{region '#Template'}
	{attribute 'Category' := 'AC'}
	{attribute 'Version' := '0.0.1.0'}
	{attribute 'Tags' := 'AC, Plant, AHU, Air handling unit'}
	{attribute 'Description' := 'Lüftungsanlage	// Air handling unit'}
{endregion}
FUNCTION_BLOCK FB_BA_AHU_1St_PrHtr_ErcPl_Col EXTENDS FB_BA_View
VAR_INPUT CONSTANT	
	TOuA					: FB_BA_SensorAnalog_IO;			
	TExhA					: FB_BA_SensorAnalog_IO;	
	TSuA					: FB_BA_SensorAnalog_IO;	
	TExtA					: FB_BA_SensorAnalog_IO;								
	TRm						: FB_BA_SensorAnalog_IO;	
	DiffPrssOuAFilt			: FB_BA_SensorAnalog_IO;											
	FiltOuAMonit			: FB_BA_Hys_21;							
	DiffPrssExtAFilt		: FB_BA_SensorAnalog_IO;				
	FiltExtAMonit			: FB_BA_Hys_21;	
	SumNgtCol				: FB_BA_AC_SumNgtCol;	
	OpMod					: FB_BA_AC_OpMod1St;	
	OuADmp					: FB_BA_Dmp2P;	
	SuAPrss					: FB_BA_SensorAnalog_IO;	
	SuADiffPrss				: FB_BA_SensorAnalog_IO;		
	SuAFan					: FB_BA_MotCtlExt;	
	SuADiffPrssMonit		: FB_BA_FdbAnalog;								
	ExhADmp					: FB_BA_Dmp2P;	
	ExtAPrss				: FB_BA_SensorAnalog_IO;	
	ExtADiffPrss			: FB_BA_SensorAnalog_IO;		
	ExtAFan					: FB_BA_MotCtlExt;								
	ExtADiffPrssMonit		: FB_BA_FdbAnalog;
	SpTRm					: FB_BA_AC_SpTRm_01;	
	TCasCtrl				: FB_BA_AC_TCasCtrl_01;										 								
	TSeqLink				: FB_BA_SequenceLink;
	PreHtr					: FB_BA_AC_PreHtr;	
	Erc						: FB_BA_AC_ErcPl_02;								
	Col						: FB_BA_AC_ColT_02;								
	PlantCtrl				: FB_BA_PlantCtrl;							
	GeneralSettings			: FB_BA_RawSubscriber;
	stGeneralSettings		: ST_BA_GeneralSettings;
END_VAR	
VAR
	PlantLock				: FB_BA_PlantLock	:= (iParent := THIS^);	
	
	PlantControlStatus   	:FB_BA_Label2x :=(iAggregate:=LblControl.PlantControl,		iFunction:=LblFunctions.Status);
	TSequenceControlStatus  :FB_BA_Label2x :=(iAggregate:=LblControl.TSequenceControl,	iFunction:=LblFunctions.Status);	
END_VAR
VAR // added by the converter: edge detectors and wires of the graphical bodies
    _w1 : ANY;
END_VAR

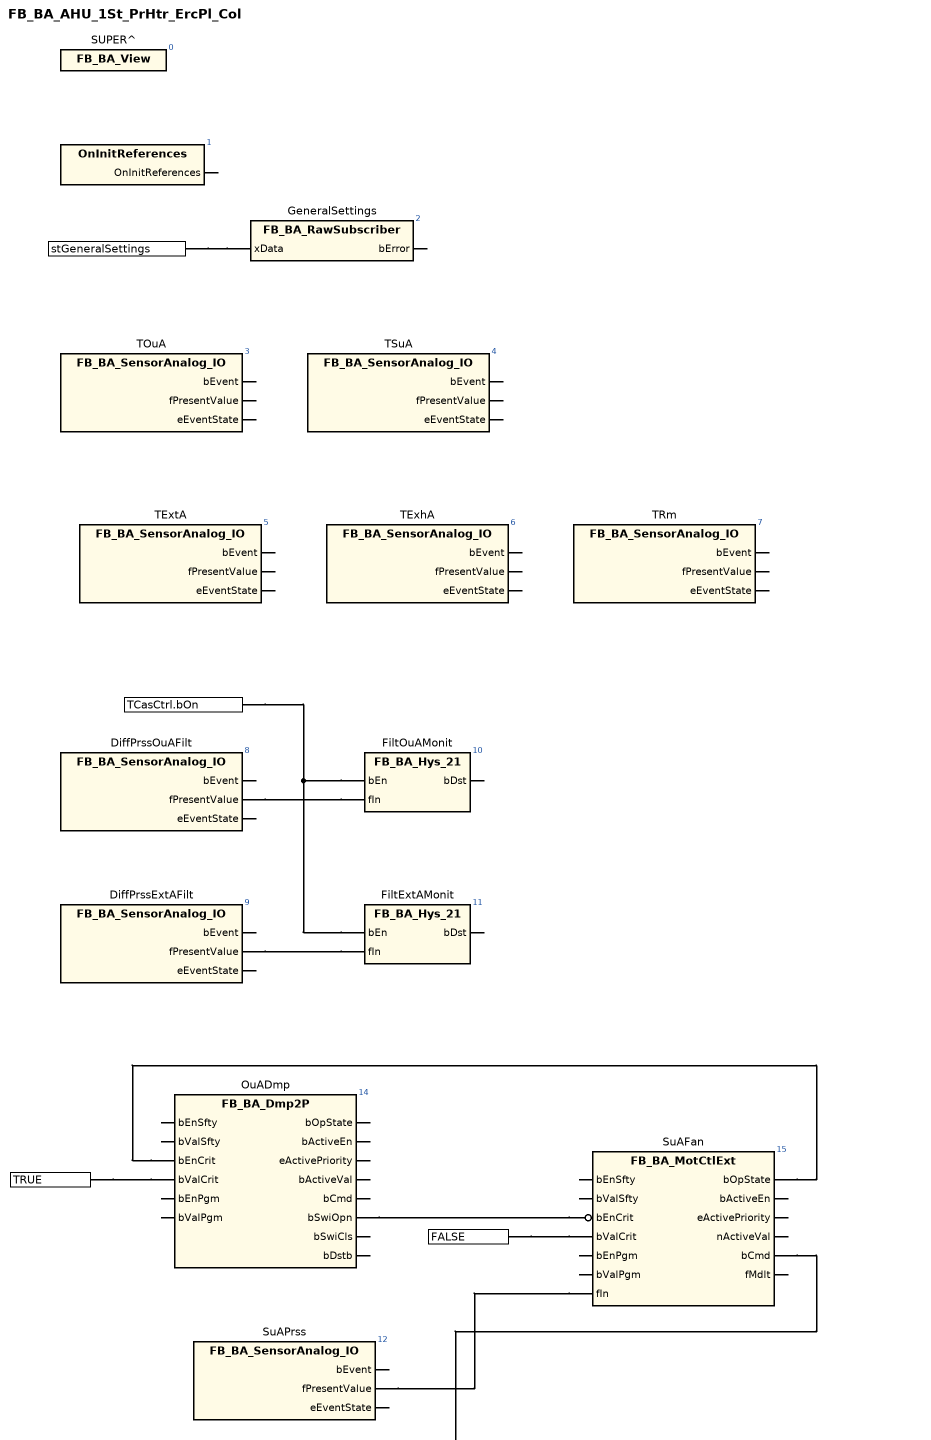
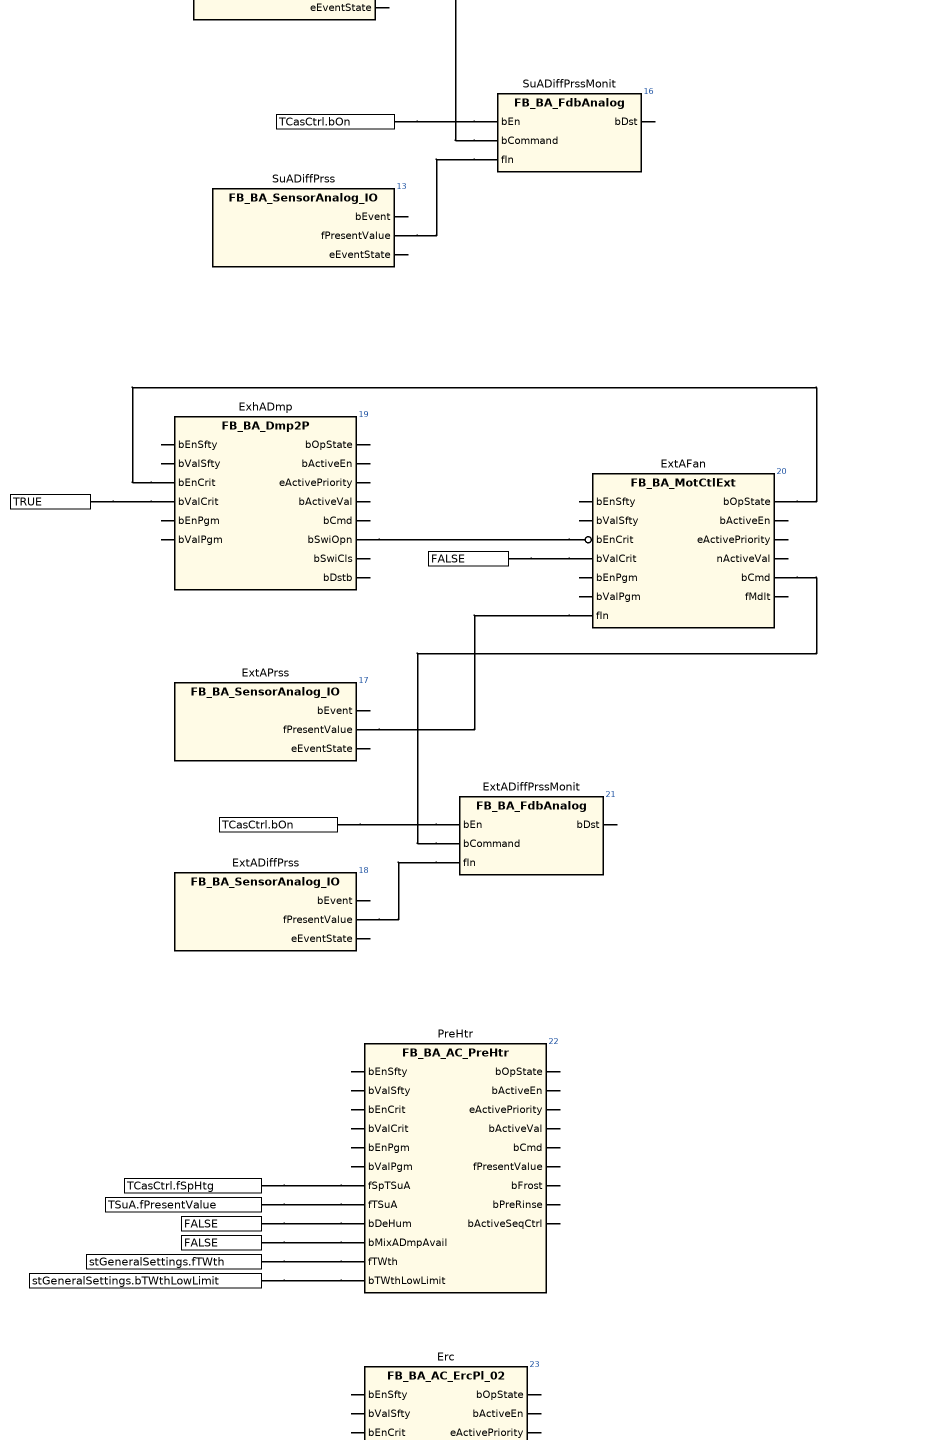
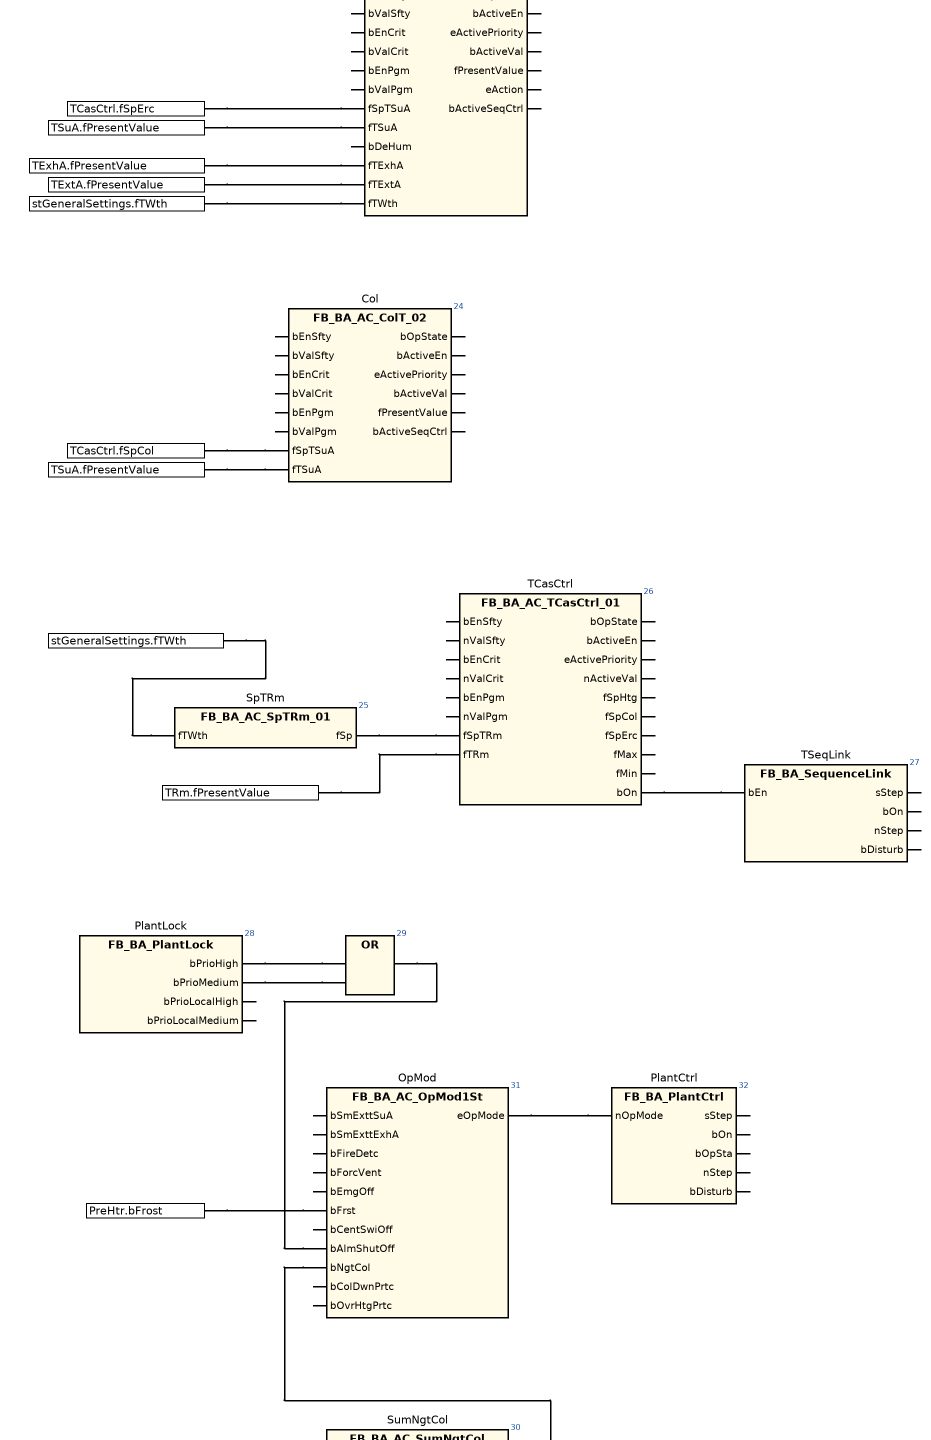
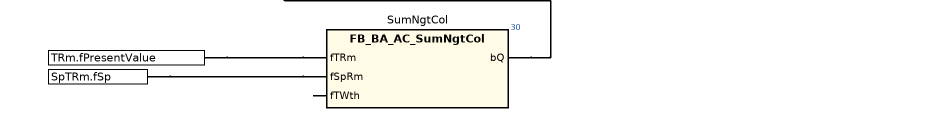
SUPER^(); // FB_BA_View
OnInitReferences();
GeneralSettings(xData := stGeneralSettings); // FB_BA_RawSubscriber
TOuA(); // FB_BA_SensorAnalog_IO
TSuA(); // FB_BA_SensorAnalog_IO
TExtA(); // FB_BA_SensorAnalog_IO
TExhA(); // FB_BA_SensorAnalog_IO
TRm(); // FB_BA_SensorAnalog_IO
DiffPrssOuAFilt(); // FB_BA_SensorAnalog_IO
DiffPrssExtAFilt(); // FB_BA_SensorAnalog_IO
FiltOuAMonit(bEn := TCasCtrl.bOn, fIn := DiffPrssOuAFilt.fPresentValue); // FB_BA_Hys_21
FiltExtAMonit(bEn := TCasCtrl.bOn, fIn := DiffPrssExtAFilt.fPresentValue); // FB_BA_Hys_21
SuAPrss(); // FB_BA_SensorAnalog_IO
SuADiffPrss(); // FB_BA_SensorAnalog_IO
OuADmp(bEnCrit := SuAFan.bOpState, bValCrit := TRUE); // FB_BA_Dmp2P
SuAFan(bEnCrit := NOT OuADmp.bSwiOpn, bValCrit := FALSE, fIn := SuAPrss.fPresentValue); // FB_BA_MotCtlExt
SuADiffPrssMonit(bEn := TCasCtrl.bOn, bCommand := SuAFan.bCmd, fIn := SuADiffPrss.fPresentValue); // FB_BA_FdbAnalog
ExtAPrss(); // FB_BA_SensorAnalog_IO
ExtADiffPrss(); // FB_BA_SensorAnalog_IO
ExhADmp(bEnCrit := ExtAFan.bOpState, bValCrit := TRUE); // FB_BA_Dmp2P
ExtAFan(bEnCrit := NOT ExhADmp.bSwiOpn, bValCrit := FALSE, fIn := ExtAPrss.fPresentValue); // FB_BA_MotCtlExt
ExtADiffPrssMonit(bEn := TCasCtrl.bOn, bCommand := ExtAFan.bCmd, fIn := ExtADiffPrss.fPresentValue); // FB_BA_FdbAnalog
PreHtr(
    fSpTSuA := TCasCtrl.fSpHtg,
    fTSuA := TSuA.fPresentValue,
    bDeHum := FALSE,
    bMixADmpAvail := FALSE,
    fTWth := stGeneralSettings.fTWth,
    bTWthLowLimit := stGeneralSettings.bTWthLowLimit); // FB_BA_AC_PreHtr
Erc(
    fSpTSuA := TCasCtrl.fSpErc,
    fTSuA := TSuA.fPresentValue,
    fTExhA := TExhA.fPresentValue,
    fTExtA := TExtA.fPresentValue,
    fTWth := stGeneralSettings.fTWth); // FB_BA_AC_ErcPl_02
Col(fSpTSuA := TCasCtrl.fSpCol, fTSuA := TSuA.fPresentValue); // FB_BA_AC_ColT_02
SpTRm(fTWth := stGeneralSettings.fTWth); // FB_BA_AC_SpTRm_01
TCasCtrl(fSpTRm := SpTRm.fSp, fTRm := TRm.fPresentValue); // FB_BA_AC_TCasCtrl_01
TSeqLink(bEn := TCasCtrl.bOn); // FB_BA_SequenceLink
PlantLock(); // FB_BA_PlantLock
_w1 := PlantLock.bPrioHigh OR PlantLock.bPrioMedium;
SumNgtCol(fTRm := TRm.fPresentValue, fSpRm := SpTRm.fSp); // FB_BA_AC_SumNgtCol
OpMod(bFrst := PreHtr.bFrost, bAlmShutOff := _w1, bNgtCol := SumNgtCol.bQ); // FB_BA_AC_OpMod1St
PlantCtrl(nOpMode := OpMod.eOpMode); // FB_BA_PlantCtrl

METHOD FB_init : BOOL
VAR_INPUT
	bInitRetains : BOOL; // if TRUE, the retain variables are initialized (warm start / cold start)
	bInCopyCode : BOOL;  // if TRUE, the instance afterwards gets moved into the copy code (online change)
END_VAR
TOuA.iParent								:= THIS^;		
TOuA.iLabel 								:= LblCmpAC.AHU_TOuA;	
TOuA.sObjectName							:= '{Idx=01}';	
TOuA.eDPADMode								:= E_BA_DPADMode.eInclude;										
TOuA.MV.eUnit								:= E_BA_Unit.eTemperature_DegreesCelsius;
TOuA.MV.eEnPlantLock						:= E_BA_LockPriority.eNoLock;
TOuA.MV.fResolution 						:= 0.01;
TOuA.MV.fScaleOffset 						:= 0; 

TExhA.iParent								:= THIS^;		
TExhA.iLabel 								:= LblCmpAC.AHU_TExhA;	
TExhA.sObjectName							:= '{Idx=01}';												
TExhA.eDPADMode								:= E_BA_DPADMode.eInclude;										
TExhA.MV.eUnit								:= E_BA_Unit.eTemperature_DegreesCelsius;
TExhA.MV.eEnPlantLock						:= E_BA_LockPriority.eNoLock;
TExhA.MV.fResolution 						:= 0.01;
TExhA.MV.fScaleOffset 						:= 0; 

TSuA.iParent								:= THIS^;		
TSuA.iLabel 								:= LblCmpAC.AHU_TSuA;	
TSuA.sObjectName							:= '{Idx=01}';
TSuA.eDPADMode								:= E_BA_DPADMode.eInclude;										
TSuA.MV.eUnit								:= E_BA_Unit.eTemperature_DegreesCelsius;
TSuA.MV.eEnPlantLock						:= E_BA_LockPriority.eMedium;
TSuA.MV.fResolution 						:= 0.01;
TSuA.MV.fScaleOffset 						:= 0; 

TExtA.iParent								:= THIS^;
TExtA.iLabel 								:= LblCmpAC.AHU_TExtA;	
TExtA.sObjectName							:= '{Idx=01}'; 
TExtA.eDPADMode								:= E_BA_DPADMode.eInclude;										
TExtA.MV.eUnit								:= E_BA_Unit.eTemperature_DegreesCelsius;
TExtA.MV.eEnPlantLock						:= E_BA_LockPriority.eNoLock;
TExtA.MV.fResolution 						:= 0.01;
TExtA.MV.fScaleOffset 						:= 0; 

TRm.iParent									:= THIS^;		
TRm.iLabel 									:= LblCmpAC.AHU_TRm;	
TRm.sObjectName								:= '{Idx=01}';
TRm.eDPADMode								:= E_BA_DPADMode.eInclude;										
TRm.MV.eUnit								:= E_BA_Unit.eTemperature_DegreesCelsius;
TRm.MV.eEnPlantLock							:= E_BA_LockPriority.eNoLock;
TRm.MV.fResolution 							:= 0.01;
TRm.MV.fScaleOffset 						:= 0;

DiffPrssOuAFilt.iParent						:= THIS^;		
DiffPrssOuAFilt.iLabel 						:= LblCmpAC.AHU_DiffPrssOuAFilt;	
DiffPrssOuAFilt.sObjectName					:= '{Idx=03}';												
DiffPrssOuAFilt.eDPADMode					:= E_BA_DPADMode.eInclude;										
DiffPrssOuAFilt.MV.eUnit					:= E_BA_Unit.ePressure_Pascals;
DiffPrssOuAFilt.MV.eEnPlantLock				:= E_BA_LockPriority.eNoLock;
DiffPrssOuAFilt.MV.fResolution 				:= 0.03051851;
DiffPrssOuAFilt.MV.fScaleOffset 			:= 0; 

FiltOuAMonit.iParent						:= THIS^;
FiltOuAMonit.iLabel							:= LblCmpAC.AHU_FiltOuAMonit;
FiltOuAMonit.sObjectName					:= '{Idx=01}';										 
FiltOuAMonit.eDPADMode						:= E_BA_DPADMode.eInclude;
FiltOuAMonit.DstMainAlarm.eEnPlantLock		:= E_BA_LockPriority.eMedium;

DiffPrssExtAFilt.iParent					:= THIS^;		
DiffPrssExtAFilt.iLabel 					:= LblCmpAC.AHU_DiffPrssExtAFilt;	
DiffPrssExtAFilt.sObjectName				:= '{Idx=04}';
DiffPrssExtAFilt.eDPADMode					:= E_BA_DPADMode.eInclude;										
DiffPrssExtAFilt.MV.eUnit					:= E_BA_Unit.ePressure_Pascals;
DiffPrssExtAFilt.MV.eEnPlantLock			:= E_BA_LockPriority.eNoLock;
DiffPrssExtAFilt.MV.fResolution 			:= 0.03051851;
DiffPrssExtAFilt.MV.fScaleOffset 			:= 0; 

FiltExtAMonit.iParent						:= THIS^;
FiltExtAMonit.iLabel						:= LblCmpAC.AHU_FiltExtAMonit;
FiltExtAMonit.sObjectName					:= '{Idx=02}';										 
FiltExtAMonit.eDPADMode						:= E_BA_DPADMode.eInclude;
FiltExtAMonit.DstMainAlarm.eEnPlantLock		:= E_BA_LockPriority.eMedium;

SumNgtCol.iParent							:= THIS^;
SumNgtCol.iLabel							:= LblCmpAC.AHU_SumNgtCol;
SumNgtCol.sObjectName						:= '{Idx=01}';										 
SumNgtCol.eDPADMode							:= E_BA_DPADMode.eInclude;								

OpMod.iParent								:= THIS^;
OpMod.iLabel								:= LblCmpAC.AHU_OpMod;
OpMod.sObjectName							:= '{Idx=01}';										 
OpMod.eDPADMode								:= E_BA_DPADMode.eInclude;								

OuADmp.iParent								:= THIS^;
OuADmp.iLabel								:= LblCmpAC.AHU_OuADmp;
OuADmp.sObjectName							:= '{Idx=01}';										 
OuADmp.eDPADMode							:= E_BA_DPADMode.eInclude;								

SuAPrss.iParent								:= THIS^;		
SuAPrss.iLabel 								:= LblCmpAC.AHU_SuAPrss;	
SuAPrss.sObjectName							:= '{Idx=01}';
SuAPrss.eDPADMode							:= E_BA_DPADMode.eInclude;																						
SuAPrss.MV.eUnit							:= E_BA_Unit.ePressure_Pascals;
SuAPrss.MV.eEnPlantLock						:= E_BA_LockPriority.eNoLock;
SuAPrss.MV.fResolution 						:= 0.03051851;
SuAPrss.MV.fScaleOffset 					:= 0;

SuADiffPrss.iParent							:= THIS^;		
SuADiffPrss.iLabel 							:= LblCmpAC.AHU_SuADiffPrss;	
SuADiffPrss.sObjectName						:= '{Idx=01}';
SuADiffPrss.eDPADMode						:= E_BA_DPADMode.eInclude;																						
SuADiffPrss.MV.eUnit						:= E_BA_Unit.ePressure_Pascals;
SuADiffPrss.MV.eEnPlantLock					:= E_BA_LockPriority.eNoLock;
SuADiffPrss.MV.fResolution 					:= 0.03051851;
SuADiffPrss.MV.fScaleOffset 				:= 0; 

SuAFan.iParent								:= THIS^;
SuAFan.iLabel								:= LblCmpAC.AHU_SuAFan;
SuAFan.sObjectName							:= '{Idx=01}';										 
SuAFan.eDPADMode							:= E_BA_DPADMode.eInclude;								

SuADiffPrssMonit.iParent					:= THIS^;
SuADiffPrssMonit.iLabel						:= LblCmpAC.AHU_SuADiffPrssMonit;
SuADiffPrssMonit.sObjectName				:= '{Idx=01}';										 
SuADiffPrssMonit.eDPADMode					:= E_BA_DPADMode.eInclude;								

ExhADmp.iParent								:= THIS^;
ExhADmp.iLabel								:= LblCmpAC.AHU_ExhADmp;
ExhADmp.sObjectName							:= '{Idx=02}';										 
ExhADmp.eDPADMode							:= E_BA_DPADMode.eInclude;								

ExtAPrss.iParent							:= THIS^;		
ExtAPrss.iLabel 							:= LblCmpAC.AHU_ExtAPrss;	
ExtAPrss.sObjectName						:= '{Idx=01}';												
ExtAPrss.eDPADMode							:= E_BA_DPADMode.eInclude;																						
ExtAPrss.MV.eUnit							:= E_BA_Unit.ePressure_Pascals;
ExtAPrss.MV.eEnPlantLock					:= E_BA_LockPriority.eNoLock;
ExtAPrss.MV.fResolution 					:= 0.03051851;
ExtAPrss.MV.fScaleOffset 					:= 0; 

ExtADiffPrss.iParent						:= THIS^;		
ExtADiffPrss.iLabel 						:= LblCmpAC.AHU_ExtADiffPrss;	
ExtADiffPrss.sObjectName					:= '{Idx=02}';
ExtADiffPrss.eDPADMode						:= E_BA_DPADMode.eInclude;																						
ExtADiffPrss.MV.eUnit						:= E_BA_Unit.ePressure_Pascals;
ExtADiffPrss.MV.eEnPlantLock				:= E_BA_LockPriority.eNoLock;
ExtADiffPrss.MV.fResolution 				:= 0.03051851;
ExtADiffPrss.MV.fScaleOffset 				:= 0; 

ExtAFan.iParent								:= THIS^;
ExtAFan.iLabel								:= LblCmpAC.AHU_ExtAFan;
ExtAFan.sObjectName							:= '{Idx=01}';										 
ExtAFan.eDPADMode							:= E_BA_DPADMode.eInclude;								

ExtADiffPrssMonit.iParent					:= THIS^;
ExtADiffPrssMonit.iLabel					:= LblCmpAC.AHU_ExtADiffPrssMonit;
ExtADiffPrssMonit.sObjectName				:= '{Idx=02}';										 
ExtADiffPrssMonit.eDPADMode					:= E_BA_DPADMode.eInclude;								

SpTRm.iParent								:= THIS^;
SpTRm.iLabel								:= LblCmpAC.AHU_SpTRm;
SpTRm.sObjectName							:= '{Idx=01}';										 
SpTRm.eDPADMode								:= E_BA_DPADMode.eInclude;								

TCasCtrl.iParent							:= THIS^;
TCasCtrl.iLabel								:= LblCmpAC.AHU_TCasCtrl;
TCasCtrl.sObjectName						:= '{Idx=01}';										 
TCasCtrl.eDPADMode							:= E_BA_DPADMode.eInclude;																		 								

TSeqLink.iParent							:= THIS^;
TSeqLink.iLabel								:= LblCmpAC.AHU_TSeqLink;
TSeqLink.sObjectName						:= '{Idx=01,Idx=01}';									
TSeqLink.iReference[1]						:= PreHtr.TSuACtrl.Ctrl;
TSeqLink.iReference[2]						:= Erc.TSuACtrl.Ctrl;
TSeqLink.iReference[3]						:= Col.TSuACtrl.Ctrl;

PreHtr.iParent								:= THIS^;
PreHtr.iLabel								:= LblCmpAC.AHU_PreHtr;
PreHtr.sObjectName							:= '{Idx=01}';										 
PreHtr.eDPADMode							:= E_BA_DPADMode.eIncludeDescription;								

Erc.iParent									:= THIS^;
Erc.iLabel									:= LblCmpAC.AHU_Erc;
Erc.sObjectName								:= '{Idx=01}';										 
Erc.eDPADMode								:= E_BA_DPADMode.eIncludeDescription;																

Col.iParent									:= THIS^;
Col.iLabel									:= LblCmpAC.AHU_Col;
Col.sObjectName								:= '{Idx=01}';										 
Col.eDPADMode								:= E_BA_DPADMode.eIncludeDescription;								

PlantCtrl.iParent							:= THIS^;
PlantCtrl.iLabel							:= LblCmpAC.AHU_PlantCtrl;
PlantCtrl.sObjectName						:= '{Idx=01,Idx=01}';
PlantCtrl.aStateText						:= OpMod.OpModPr.aStateText;	

GeneralSettings.Subject						:= Site.GeneralSettings_Subject;
GeneralSettings.sTarget						:= Site.GeneralSettings_NetId;
END_METHOD

METHOD Init_OffOn : BOOL
// Apply configured states:
(*

WIRD DIESE DEKLARATION HIER BENÖTIGT????
23.02.2021 FP

OpMod.OpModMan.aStateText[1] := Texts.txtAuto;
OpMod.OpModMan.aStateText[2] := Texts.txtOff;
OpMod.OpModMan.aStateText[3] := Texts.txtOn;

OpMod.Sched.aStateText[1] := Texts.txtOff;
OpMod.Sched.aStateText[2] := Texts.txtOn;

OpMod.OpModPr.aStateText[1]		:= Texts.txtOff;
OpMod.OpModPr.aStateText[2]		:= Texts.txtOn;
OpMod.OpModPr.aStateText[3]		:= Texts.txtEmergencyStop;
OpMod.OpModPr.aStateText[4]		:= Texts.txtFrost;
OpMod.OpModPr.aStateText[5]		:= Texts.txtSmokeExtraction_P;
OpMod.OpModPr.aStateText[6]		:= Texts.txtSmokeExtractionSupplyAir;
OpMod.OpModPr.aStateText[7]		:= Texts.txtSmokeExtractionExtractAir;
OpMod.OpModPr.aStateText[8]		:= Texts.txtFire;
OpMod.OpModPr.aStateText[9]		:= Texts.txtNightCooling;
OpMod.OpModPr.aStateText[10]	:= Texts.txtCoolDownProtection;
OpMod.OpModPr.aStateText[11]	:= Texts.txtOverHeatingProtection;
OpMod.OpModPr.aStateText[12]	:= Texts.txtDisturb;
OpMod.OpModPr.aStateText[13]	:= Texts.txtForcedVentilation;
OpMod.OpModPr.aStateText[14]	:= Texts.txtCentralSwitchOff;
*)

// plant operations modes with priorities:
PlantCtrl.AddOperationMode(nOpMode := E_BA_AC_OpMod01.eOff,							ePriority := E_BA_Priority.eProgram);
PlantCtrl.AddOperationMode(nOpMode := E_BA_AC_OpMod01.eOn,							ePriority := E_BA_Priority.eProgram);
PlantCtrl.AddOperationMode(nOpMode := E_BA_AC_OpMod01.eNightCooling,				ePriority := E_BA_Priority.eProgram);
PlantCtrl.AddOperationMode(nOpMode := E_BA_AC_OpMod01.eCoolDownProtection,			ePriority := E_BA_Priority.eProgram);
PlantCtrl.AddOperationMode(nOpMode := E_BA_AC_OpMod01.eOverHeatingProtection,		ePriority := E_BA_Priority.eProgram);
PlantCtrl.AddOperationMode(nOpMode := E_BA_AC_OpMod01.eFrost,						ePriority := E_BA_Priority.eCritical);
PlantCtrl.AddOperationMode(nOpMode := E_BA_AC_OpMod01.eEmergency,					ePriority := E_BA_Priority.eCritical);
PlantCtrl.AddOperationMode(nOpMode := E_BA_AC_OpMod01.eAlarm,						ePriority := E_BA_Priority.eCritical);
PlantCtrl.AddOperationMode(nOpMode := E_BA_AC_OpMod01.eForcedVentilation,			ePriority := E_BA_Priority.eCritical);
PlantCtrl.AddOperationMode(nOpMode := E_BA_AC_OpMod01.eCentralSwitchOff,			ePriority := E_BA_Priority.eCritical);
PlantCtrl.AddOperationMode(nOpMode := E_BA_AC_OpMod01.eSmokeExtractionProgramm,		ePriority := E_BA_Priority.eLifeSafety);
PlantCtrl.AddOperationMode(nOpMode := E_BA_AC_OpMod01.eSmokeExtractionSupplyAir,	ePriority := E_BA_Priority.eLifeSafety);
PlantCtrl.AddOperationMode(nOpMode := E_BA_AC_OpMod01.eSmokeExtractionExhaustAir,	ePriority := E_BA_Priority.eLifeSafety);
PlantCtrl.AddOperationMode(nOpMode := E_BA_AC_OpMod01.eFire, 						ePriority := E_BA_Priority.eLifeSafety);

// Start sequence Step order and parameter
PlantCtrl.AddAggregate(iReference := PreHtr,	bWaitForProcesses := TRUE,	bWaitForEvents := FALSE, tDelayStepDown := T#0S, tDelayStepUp := T#5S);
PlantCtrl.AddAggregate(iReference := OuADmp,	bWaitForProcesses := FALSE, bWaitForEvents := FALSE, tDelayStepDown := T#2S, tDelayStepUp := T#2S);
PlantCtrl.AddAggregate(iReference := ExhADmp,	bWaitForProcesses := FALSE, bWaitForEvents := FALSE, tDelayStepDown := T#2S, tDelayStepUp := T#2S);
PlantCtrl.AddAggregate(iReference := SuAFan,	bWaitForProcesses := FALSE, bWaitForEvents := FALSE, tDelayStepDown := T#2S, tDelayStepUp := T#2S);
PlantCtrl.AddAggregate(iReference := ExtAFan,	bWaitForProcesses := FALSE, bWaitForEvents := FALSE, tDelayStepDown := T#2S, tDelayStepUp := T#2S);
PlantCtrl.AddAggregate(iReference := Erc,		bWaitForProcesses := FALSE, bWaitForEvents := FALSE, tDelayStepDown := T#0S, tDelayStepUp := T#0S);
PlantCtrl.AddAggregate(iReference := Col,		bWaitForProcesses := FALSE, bWaitForEvents := FALSE, tDelayStepDown := T#0S, tDelayStepUp := T#0S);
PlantCtrl.AddAggregate(iReference := TCasCtrl,	bWaitForProcesses := FALSE, bWaitForEvents := FALSE, tDelayStepDown := T#0S, tDelayStepUp := T#0S);

// Apply aggregate operation modes dependant on corresponding plant operation modes:
// [Controlling aggregates]
// release pre-heater depending on plant operation mode 
PlantCtrl.AssignAggregate1x(nPltOpMode := E_BA_AC_OpMod01.eOff,							iAgg1Ref := PreHtr, nAgg1OpMode := TO_UDINT(FALSE));
PlantCtrl.AssignAggregate1x(nPltOpMode := E_BA_AC_OpMod01.eOn,							iAgg1Ref := PreHtr, nAgg1OpMode := TO_UDINT(TRUE));
PlantCtrl.AssignAggregate1x(nPltOpMode := E_BA_AC_OpMod01.eNightCooling,				iAgg1Ref := PreHtr, nAgg1OpMode := TO_UDINT(FALSE));
PlantCtrl.AssignAggregate1x(nPltOpMode := E_BA_AC_OpMod01.eCoolDownProtection,			iAgg1Ref := PreHtr, nAgg1OpMode := TO_UDINT(TRUE));
PlantCtrl.AssignAggregate1x(nPltOpMode := E_BA_AC_OpMod01.eOverHeatingProtection,		iAgg1Ref := PreHtr, nAgg1OpMode := TO_UDINT(FALSE));
PlantCtrl.AssignAggregate1x(nPltOpMode := E_BA_AC_OpMod01.eFrost,						iAgg1Ref := PreHtr, nAgg1OpMode := TO_UDINT(TRUE));
PlantCtrl.AssignAggregate1x(nPltOpMode := E_BA_AC_OpMod01.eEmergency,					iAgg1Ref := PreHtr, nAgg1OpMode := TO_UDINT(FALSE));
PlantCtrl.AssignAggregate1x(nPltOpMode := E_BA_AC_OpMod01.eAlarm,						iAgg1Ref := PreHtr, nAgg1OpMode := TO_UDINT(FALSE));
PlantCtrl.AssignAggregate1x(nPltOpMode := E_BA_AC_OpMod01.eForcedVentilation,			iAgg1Ref := PreHtr, nAgg1OpMode := TO_UDINT(TRUE));
PlantCtrl.AssignAggregate1x(nPltOpMode := E_BA_AC_OpMod01.eCentralSwitchOff,			iAgg1Ref := PreHtr, nAgg1OpMode := TO_UDINT(FALSE));
PlantCtrl.AssignAggregate1x(nPltOpMode := E_BA_AC_OpMod01.eSmokeExtractionProgramm,		iAgg1Ref := PreHtr, nAgg1OpMode := TO_UDINT(TRUE));
PlantCtrl.AssignAggregate1x(nPltOpMode := E_BA_AC_OpMod01.eSmokeExtractionSupplyAir,	iAgg1Ref := PreHtr, nAgg1OpMode := TO_UDINT(TRUE));
PlantCtrl.AssignAggregate1x(nPltOpMode := E_BA_AC_OpMod01.eSmokeExtractionExhaustAir,	iAgg1Ref := PreHtr, nAgg1OpMode := TO_UDINT(FALSE));
PlantCtrl.AssignAggregate1x(nPltOpMode := E_BA_AC_OpMod01.eFire,						iAgg1Ref := PreHtr, nAgg1OpMode := TO_UDINT(FALSE));

// Apply aggregate operation modes dependant on corresponding plant operation modes:
// [Controlling aggregates]
// release Erc depending on plant operation mode 
PlantCtrl.AssignAggregate1x(nPltOpMode := E_BA_AC_OpMod01.eOff,							iAgg1Ref := Erc, nAgg1OpMode := TO_UDINT(FALSE));
PlantCtrl.AssignAggregate1x(nPltOpMode := E_BA_AC_OpMod01.eOn,							iAgg1Ref := Erc, nAgg1OpMode := TO_UDINT(TRUE));
PlantCtrl.AssignAggregate1x(nPltOpMode := E_BA_AC_OpMod01.eNightCooling,				iAgg1Ref := Erc, nAgg1OpMode := TO_UDINT(FALSE));
PlantCtrl.AssignAggregate1x(nPltOpMode := E_BA_AC_OpMod01.eCoolDownProtection,			iAgg1Ref := Erc, nAgg1OpMode := TO_UDINT(TRUE));
PlantCtrl.AssignAggregate1x(nPltOpMode := E_BA_AC_OpMod01.eOverHeatingProtection,		iAgg1Ref := Erc, nAgg1OpMode := TO_UDINT(TRUE));
PlantCtrl.AssignAggregate1x(nPltOpMode := E_BA_AC_OpMod01.eFrost,						iAgg1Ref := Erc, nAgg1OpMode := TO_UDINT(TRUE));
PlantCtrl.AssignAggregate1x(nPltOpMode := E_BA_AC_OpMod01.eEmergency,					iAgg1Ref := Erc, nAgg1OpMode := TO_UDINT(FALSE));
PlantCtrl.AssignAggregate1x(nPltOpMode := E_BA_AC_OpMod01.eAlarm,						iAgg1Ref := Erc, nAgg1OpMode := TO_UDINT(FALSE));
PlantCtrl.AssignAggregate1x(nPltOpMode := E_BA_AC_OpMod01.eForcedVentilation,			iAgg1Ref := Erc, nAgg1OpMode := TO_UDINT(TRUE));
PlantCtrl.AssignAggregate1x(nPltOpMode := E_BA_AC_OpMod01.eCentralSwitchOff,			iAgg1Ref := Erc, nAgg1OpMode := TO_UDINT(FALSE));
PlantCtrl.AssignAggregate1x(nPltOpMode := E_BA_AC_OpMod01.eSmokeExtractionProgramm,		iAgg1Ref := Erc, nAgg1OpMode := TO_UDINT(TRUE));
PlantCtrl.AssignAggregate1x(nPltOpMode := E_BA_AC_OpMod01.eSmokeExtractionSupplyAir,	iAgg1Ref := Erc, nAgg1OpMode := TO_UDINT(TRUE));
PlantCtrl.AssignAggregate1x(nPltOpMode := E_BA_AC_OpMod01.eSmokeExtractionExhaustAir,	iAgg1Ref := Erc, nAgg1OpMode := TO_UDINT(TRUE));
PlantCtrl.AssignAggregate1x(nPltOpMode := E_BA_AC_OpMod01.eFire,						iAgg1Ref := Erc, nAgg1OpMode := TO_UDINT(FALSE));

// Apply aggregate operation modes dependant on corresponding plant operation modes:
// [Controlling aggregates]
// release cooler depending on plant operation mode 
PlantCtrl.AssignAggregate1x(nPltOpMode := E_BA_AC_OpMod01.eOff,							iAgg1Ref := Col, nAgg1OpMode := TO_UDINT(FALSE));
PlantCtrl.AssignAggregate1x(nPltOpMode := E_BA_AC_OpMod01.eOn,							iAgg1Ref := Col, nAgg1OpMode := TO_UDINT(TRUE));
PlantCtrl.AssignAggregate1x(nPltOpMode := E_BA_AC_OpMod01.eNightCooling,				iAgg1Ref := Col, nAgg1OpMode := TO_UDINT(FALSE));
PlantCtrl.AssignAggregate1x(nPltOpMode := E_BA_AC_OpMod01.eCoolDownProtection,			iAgg1Ref := Col, nAgg1OpMode := TO_UDINT(FALSE));
PlantCtrl.AssignAggregate1x(nPltOpMode := E_BA_AC_OpMod01.eOverHeatingProtection,		iAgg1Ref := Col, nAgg1OpMode := TO_UDINT(TRUE));
PlantCtrl.AssignAggregate1x(nPltOpMode := E_BA_AC_OpMod01.eFrost,						iAgg1Ref := Col, nAgg1OpMode := TO_UDINT(FALSE));
PlantCtrl.AssignAggregate1x(nPltOpMode := E_BA_AC_OpMod01.eEmergency,					iAgg1Ref := Col, nAgg1OpMode := TO_UDINT(FALSE));
PlantCtrl.AssignAggregate1x(nPltOpMode := E_BA_AC_OpMod01.eAlarm,						iAgg1Ref := Col, nAgg1OpMode := TO_UDINT(FALSE));
PlantCtrl.AssignAggregate1x(nPltOpMode := E_BA_AC_OpMod01.eForcedVentilation,			iAgg1Ref := Col, nAgg1OpMode := TO_UDINT(TRUE));
PlantCtrl.AssignAggregate1x(nPltOpMode := E_BA_AC_OpMod01.eCentralSwitchOff,			iAgg1Ref := Col, nAgg1OpMode := TO_UDINT(FALSE));
PlantCtrl.AssignAggregate1x(nPltOpMode := E_BA_AC_OpMod01.eSmokeExtractionProgramm,		iAgg1Ref := Col, nAgg1OpMode := TO_UDINT(FALSE));
PlantCtrl.AssignAggregate1x(nPltOpMode := E_BA_AC_OpMod01.eSmokeExtractionSupplyAir,	iAgg1Ref := Col, nAgg1OpMode := TO_UDINT(FALSE));
PlantCtrl.AssignAggregate1x(nPltOpMode := E_BA_AC_OpMod01.eSmokeExtractionExhaustAir,	iAgg1Ref := Col, nAgg1OpMode := TO_UDINT(FALSE));
PlantCtrl.AssignAggregate1x(nPltOpMode := E_BA_AC_OpMod01.eFire,						iAgg1Ref := Col, nAgg1OpMode := TO_UDINT(FALSE));

// Apply aggregate operation modes dependant on corresponding plant operation modes:
// [Controlling aggregates]
// [Outside air damper]
PlantCtrl.AssignAggregate1x(nPltOpMode := E_BA_AC_OpMod01.eOff,							iAgg1Ref := OuADmp, nAgg1OpMode := TO_UDINT(FALSE));
PlantCtrl.AssignAggregate1x(nPltOpMode := E_BA_AC_OpMod01.eOn,							iAgg1Ref := OuADmp, nAgg1OpMode := TO_UDINT(TRUE));
PlantCtrl.AssignAggregate1x(nPltOpMode := E_BA_AC_OpMod01.eNightCooling,				iAgg1Ref := OuADmp, nAgg1OpMode := TO_UDINT(TRUE));
PlantCtrl.AssignAggregate1x(nPltOpMode := E_BA_AC_OpMod01.eCoolDownProtection,			iAgg1Ref := OuADmp, nAgg1OpMode := TO_UDINT(TRUE));
PlantCtrl.AssignAggregate1x(nPltOpMode := E_BA_AC_OpMod01.eOverHeatingProtection,		iAgg1Ref := OuADmp, nAgg1OpMode := TO_UDINT(TRUE));
PlantCtrl.AssignAggregate1x(nPltOpMode := E_BA_AC_OpMod01.eFrost,						iAgg1Ref := OuADmp, nAgg1OpMode := TO_UDINT(FALSE));
PlantCtrl.AssignAggregate1x(nPltOpMode := E_BA_AC_OpMod01.eEmergency,					iAgg1Ref := OuADmp, nAgg1OpMode := TO_UDINT(FALSE));
PlantCtrl.AssignAggregate1x(nPltOpMode := E_BA_AC_OpMod01.eAlarm,						iAgg1Ref := OuADmp, nAgg1OpMode := TO_UDINT(FALSE));
PlantCtrl.AssignAggregate1x(nPltOpMode := E_BA_AC_OpMod01.eForcedVentilation,			iAgg1Ref := OuADmp, nAgg1OpMode := TO_UDINT(TRUE));
PlantCtrl.AssignAggregate1x(nPltOpMode := E_BA_AC_OpMod01.eCentralSwitchOff,			iAgg1Ref := OuADmp, nAgg1OpMode := TO_UDINT(FALSE));
PlantCtrl.AssignAggregate1x(nPltOpMode := E_BA_AC_OpMod01.eSmokeExtractionProgramm,		iAgg1Ref := OuADmp, nAgg1OpMode := TO_UDINT(TRUE));
PlantCtrl.AssignAggregate1x(nPltOpMode := E_BA_AC_OpMod01.eSmokeExtractionSupplyAir,	iAgg1Ref := OuADmp, nAgg1OpMode := TO_UDINT(TRUE));
PlantCtrl.AssignAggregate1x(nPltOpMode := E_BA_AC_OpMod01.eSmokeExtractionExhaustAir,	iAgg1Ref := OuADmp, nAgg1OpMode := TO_UDINT(FALSE));
PlantCtrl.AssignAggregate1x(nPltOpMode := E_BA_AC_OpMod01.eFire,						iAgg1Ref := OuADmp, nAgg1OpMode := TO_UDINT(FALSE));

// Apply aggregate operation modes dependant on corresponding plant operation modes:
// [Controlling aggregates]
// [supply air fan]
PlantCtrl.AssignAggregate1x(nPltOpMode := E_BA_AC_OpMod01.eOff,							iAgg1Ref := SuAFan, nAgg1OpMode := E_BA_MdltCmd.eOff);
PlantCtrl.AssignAggregate1x(nPltOpMode := E_BA_AC_OpMod01.eOn,							iAgg1Ref := SuAFan, nAgg1OpMode := E_BA_MdltCmd.eOn);
PlantCtrl.AssignAggregate1x(nPltOpMode := E_BA_AC_OpMod01.eNightCooling,				iAgg1Ref := SuAFan, nAgg1OpMode := E_BA_MdltCmd.eOn);
PlantCtrl.AssignAggregate1x(nPltOpMode := E_BA_AC_OpMod01.eCoolDownProtection,			iAgg1Ref := SuAFan, nAgg1OpMode := E_BA_MdltCmd.eOn);
PlantCtrl.AssignAggregate1x(nPltOpMode := E_BA_AC_OpMod01.eOverHeatingProtection,		iAgg1Ref := SuAFan, nAgg1OpMode := E_BA_MdltCmd.eOn);
PlantCtrl.AssignAggregate1x(nPltOpMode := E_BA_AC_OpMod01.eFrost,						iAgg1Ref := SuAFan, nAgg1OpMode := E_BA_MdltCmd.eOff);
PlantCtrl.AssignAggregate1x(nPltOpMode := E_BA_AC_OpMod01.eEmergency,					iAgg1Ref := SuAFan, nAgg1OpMode := E_BA_MdltCmd.eOff);
PlantCtrl.AssignAggregate1x(nPltOpMode := E_BA_AC_OpMod01.eAlarm,						iAgg1Ref := SuAFan, nAgg1OpMode := E_BA_MdltCmd.eOff);
PlantCtrl.AssignAggregate1x(nPltOpMode := E_BA_AC_OpMod01.eForcedVentilation,			iAgg1Ref := SuAFan, nAgg1OpMode := E_BA_MdltCmd.eOn);
PlantCtrl.AssignAggregate1x(nPltOpMode := E_BA_AC_OpMod01.eCentralSwitchOff,			iAgg1Ref := SuAFan, nAgg1OpMode := E_BA_MdltCmd.eOff);
PlantCtrl.AssignAggregate1x(nPltOpMode := E_BA_AC_OpMod01.eSmokeExtractionProgramm,		iAgg1Ref := SuAFan, nAgg1OpMode := E_BA_MdltCmd.eOn);
PlantCtrl.AssignAggregate1x(nPltOpMode := E_BA_AC_OpMod01.eSmokeExtractionSupplyAir,	iAgg1Ref := SuAFan, nAgg1OpMode := E_BA_MdltCmd.eOn);
PlantCtrl.AssignAggregate1x(nPltOpMode := E_BA_AC_OpMod01.eSmokeExtractionExhaustAir,	iAgg1Ref := SuAFan, nAgg1OpMode := E_BA_MdltCmd.eOff);
PlantCtrl.AssignAggregate1x(nPltOpMode := E_BA_AC_OpMod01.eFire,						iAgg1Ref := SuAFan, nAgg1OpMode := E_BA_MdltCmd.eOff);

// Apply aggregate operation modes dependant on corresponding plant operation modes:
// [Controlling aggregates]
// [exhaust air damper]
PlantCtrl.AssignAggregate1x(nPltOpMode := E_BA_AC_OpMod01.eOff,							iAgg1Ref := ExhADmp, nAgg1OpMode := TO_UDINT(FALSE));
PlantCtrl.AssignAggregate1x(nPltOpMode := E_BA_AC_OpMod01.eOn,							iAgg1Ref := ExhADmp, nAgg1OpMode := TO_UDINT(TRUE));
PlantCtrl.AssignAggregate1x(nPltOpMode := E_BA_AC_OpMod01.eNightCooling,				iAgg1Ref := ExhADmp, nAgg1OpMode := TO_UDINT(TRUE));
PlantCtrl.AssignAggregate1x(nPltOpMode := E_BA_AC_OpMod01.eCoolDownProtection,			iAgg1Ref := ExhADmp, nAgg1OpMode := TO_UDINT(TRUE));
PlantCtrl.AssignAggregate1x(nPltOpMode := E_BA_AC_OpMod01.eOverHeatingProtection,		iAgg1Ref := ExhADmp, nAgg1OpMode := TO_UDINT(TRUE));
PlantCtrl.AssignAggregate1x(nPltOpMode := E_BA_AC_OpMod01.eFrost,						iAgg1Ref := ExhADmp, nAgg1OpMode := TO_UDINT(FALSE));
PlantCtrl.AssignAggregate1x(nPltOpMode := E_BA_AC_OpMod01.eEmergency,					iAgg1Ref := ExhADmp, nAgg1OpMode := TO_UDINT(FALSE));
PlantCtrl.AssignAggregate1x(nPltOpMode := E_BA_AC_OpMod01.eAlarm,						iAgg1Ref := ExhADmp, nAgg1OpMode := TO_UDINT(FALSE));
PlantCtrl.AssignAggregate1x(nPltOpMode := E_BA_AC_OpMod01.eForcedVentilation,			iAgg1Ref := ExhADmp, nAgg1OpMode := TO_UDINT(TRUE));
PlantCtrl.AssignAggregate1x(nPltOpMode := E_BA_AC_OpMod01.eCentralSwitchOff,			iAgg1Ref := ExhADmp, nAgg1OpMode := TO_UDINT(FALSE));
PlantCtrl.AssignAggregate1x(nPltOpMode := E_BA_AC_OpMod01.eSmokeExtractionProgramm,		iAgg1Ref := ExhADmp, nAgg1OpMode := TO_UDINT(TRUE));
PlantCtrl.AssignAggregate1x(nPltOpMode := E_BA_AC_OpMod01.eSmokeExtractionSupplyAir,	iAgg1Ref := ExhADmp, nAgg1OpMode := TO_UDINT(FALSE));
PlantCtrl.AssignAggregate1x(nPltOpMode := E_BA_AC_OpMod01.eSmokeExtractionExhaustAir,	iAgg1Ref := ExhADmp, nAgg1OpMode := TO_UDINT(TRUE));
PlantCtrl.AssignAggregate1x(nPltOpMode := E_BA_AC_OpMod01.eFire,						iAgg1Ref := ExhADmp, nAgg1OpMode := TO_UDINT(FALSE));

// Apply aggregate operation modes dependant on corresponding plant operation modes:
// [Controlling aggregates]
// [exhaust air fan]
PlantCtrl.AssignAggregate1x(nPltOpMode := E_BA_AC_OpMod01.eOff,							iAgg1Ref := ExtAFan, nAgg1OpMode := E_BA_MdltCmd.eOff);
PlantCtrl.AssignAggregate1x(nPltOpMode := E_BA_AC_OpMod01.eOn,							iAgg1Ref := ExtAFan, nAgg1OpMode := E_BA_MdltCmd.eOn); 
PlantCtrl.AssignAggregate1x(nPltOpMode := E_BA_AC_OpMod01.eNightCooling,				iAgg1Ref := ExtAFan, nAgg1OpMode := E_BA_MdltCmd.eOn); 
PlantCtrl.AssignAggregate1x(nPltOpMode := E_BA_AC_OpMod01.eCoolDownProtection,			iAgg1Ref := ExtAFan, nAgg1OpMode := E_BA_MdltCmd.eOn); 
PlantCtrl.AssignAggregate1x(nPltOpMode := E_BA_AC_OpMod01.eOverHeatingProtection,		iAgg1Ref := ExtAFan, nAgg1OpMode := E_BA_MdltCmd.eOn); 
PlantCtrl.AssignAggregate1x(nPltOpMode := E_BA_AC_OpMod01.eFrost,						iAgg1Ref := ExtAFan, nAgg1OpMode := E_BA_MdltCmd.eOff);
PlantCtrl.AssignAggregate1x(nPltOpMode := E_BA_AC_OpMod01.eEmergency,					iAgg1Ref := ExtAFan, nAgg1OpMode := E_BA_MdltCmd.eOff);
PlantCtrl.AssignAggregate1x(nPltOpMode := E_BA_AC_OpMod01.eAlarm,						iAgg1Ref := ExtAFan, nAgg1OpMode := E_BA_MdltCmd.eOff);
PlantCtrl.AssignAggregate1x(nPltOpMode := E_BA_AC_OpMod01.eForcedVentilation,			iAgg1Ref := ExtAFan, nAgg1OpMode := E_BA_MdltCmd.eOn); 
PlantCtrl.AssignAggregate1x(nPltOpMode := E_BA_AC_OpMod01.eCentralSwitchOff,			iAgg1Ref := ExtAFan, nAgg1OpMode := E_BA_MdltCmd.eOff);
PlantCtrl.AssignAggregate1x(nPltOpMode := E_BA_AC_OpMod01.eSmokeExtractionProgramm,		iAgg1Ref := ExtAFan, nAgg1OpMode := E_BA_MdltCmd.eOn); 
PlantCtrl.AssignAggregate1x(nPltOpMode := E_BA_AC_OpMod01.eSmokeExtractionSupplyAir,	iAgg1Ref := ExtAFan, nAgg1OpMode := E_BA_MdltCmd.eOff);
PlantCtrl.AssignAggregate1x(nPltOpMode := E_BA_AC_OpMod01.eSmokeExtractionExhaustAir,	iAgg1Ref := ExtAFan, nAgg1OpMode := E_BA_MdltCmd.eOn); 
PlantCtrl.AssignAggregate1x(nPltOpMode := E_BA_AC_OpMod01.eFire,						iAgg1Ref := ExtAFan, nAgg1OpMode := E_BA_MdltCmd.eOff);

// Apply aggregate operation modes dependant on corresponding plant operation modes:
// [Controlling aggregates]
// [TCasCtrl]
PlantCtrl.AssignAggregate1x(nPltOpMode := E_BA_AC_OpMod01.eOff,							iAgg1Ref := TCasCtrl, nAgg1OpMode := E_BA_MdltCmd.eOff);
PlantCtrl.AssignAggregate1x(nPltOpMode := E_BA_AC_OpMod01.eOn,							iAgg1Ref := TCasCtrl, nAgg1OpMode := E_BA_MdltCmd.eOn);
PlantCtrl.AssignAggregate1x(nPltOpMode := E_BA_AC_OpMod01.eNightCooling,				iAgg1Ref := TCasCtrl, nAgg1OpMode := E_BA_MdltCmd.eOff);
PlantCtrl.AssignAggregate1x(nPltOpMode := E_BA_AC_OpMod01.eCoolDownProtection,			iAgg1Ref := TCasCtrl, nAgg1OpMode := E_BA_MdltCmd.eMax);
PlantCtrl.AssignAggregate1x(nPltOpMode := E_BA_AC_OpMod01.eOverHeatingProtection,		iAgg1Ref := TCasCtrl, nAgg1OpMode := E_BA_MdltCmd.eMin);
PlantCtrl.AssignAggregate1x(nPltOpMode := E_BA_AC_OpMod01.eFrost,						iAgg1Ref := TCasCtrl, nAgg1OpMode := E_BA_MdltCmd.eOff);
PlantCtrl.AssignAggregate1x(nPltOpMode := E_BA_AC_OpMod01.eEmergency,					iAgg1Ref := TCasCtrl, nAgg1OpMode := E_BA_MdltCmd.eOff);
PlantCtrl.AssignAggregate1x(nPltOpMode := E_BA_AC_OpMod01.eAlarm,						iAgg1Ref := TCasCtrl, nAgg1OpMode := E_BA_MdltCmd.eOff);
PlantCtrl.AssignAggregate1x(nPltOpMode := E_BA_AC_OpMod01.eForcedVentilation,			iAgg1Ref := TCasCtrl, nAgg1OpMode := E_BA_MdltCmd.eOn);
PlantCtrl.AssignAggregate1x(nPltOpMode := E_BA_AC_OpMod01.eCentralSwitchOff,			iAgg1Ref := TCasCtrl, nAgg1OpMode := E_BA_MdltCmd.eMin);
PlantCtrl.AssignAggregate1x(nPltOpMode := E_BA_AC_OpMod01.eSmokeExtractionProgramm,		iAgg1Ref := TCasCtrl, nAgg1OpMode := E_BA_MdltCmd.eMin);
PlantCtrl.AssignAggregate1x(nPltOpMode := E_BA_AC_OpMod01.eSmokeExtractionSupplyAir,	iAgg1Ref := TCasCtrl, nAgg1OpMode := E_BA_MdltCmd.eMin);
PlantCtrl.AssignAggregate1x(nPltOpMode := E_BA_AC_OpMod01.eSmokeExtractionExhaustAir,	iAgg1Ref := TCasCtrl, nAgg1OpMode := E_BA_MdltCmd.eOff);
PlantCtrl.AssignAggregate1x(nPltOpMode := E_BA_AC_OpMod01.eFire,						iAgg1Ref := TCasCtrl, nAgg1OpMode := E_BA_MdltCmd.eOff);
END_METHOD

METHOD Init_OffStep1to3 : BOOL
(*

WIRD DIESE DEKLARATION HIER BENÖTIGT????
23.02.2021 FP
// Apply configured states:
OpMod.OpModMan.aStateText := Texts.mst_Auto_Off_Step1to3;
OpMod.Sched.aStateText := Texts.mst_Off_Stept1to3;
OpMod.OpModPr.aStateText:= Texts.mst_OpMod02;
*)


// Add plant operations modes:
PlantCtrl.AddOperationMode(nOpMode := E_BA_AC_OpMod02.eOff,							ePriority := E_BA_Priority.eProgram);
PlantCtrl.AddOperationMode(nOpMode := E_BA_AC_OpMod02.eStep1,						ePriority := E_BA_Priority.eProgram);
PlantCtrl.AddOperationMode(nOpMode := E_BA_AC_OpMod02.eStep2,						ePriority := E_BA_Priority.eProgram);
PlantCtrl.AddOperationMode(nOpMode := E_BA_AC_OpMod02.eStep3,						ePriority := E_BA_Priority.eProgram);
PlantCtrl.AddOperationMode(nOpMode := E_BA_AC_OpMod02.eNightCooling,				ePriority := E_BA_Priority.eProgram);
PlantCtrl.AddOperationMode(nOpMode := E_BA_AC_OpMod02.eCoolDownProtection,			ePriority := E_BA_Priority.eProgram);
PlantCtrl.AddOperationMode(nOpMode := E_BA_AC_OpMod02.eOverHeatingProtection,		ePriority := E_BA_Priority.eProgram);
PlantCtrl.AddOperationMode(nOpMode := E_BA_AC_OpMod02.eFrost,						ePriority := E_BA_Priority.eCritical);
PlantCtrl.AddOperationMode(nOpMode := E_BA_AC_OpMod02.eEmergency,					ePriority := E_BA_Priority.eCritical);
PlantCtrl.AddOperationMode(nOpMode := E_BA_AC_OpMod02.eAlarm,						ePriority := E_BA_Priority.eCritical);
PlantCtrl.AddOperationMode(nOpMode := E_BA_AC_OpMod02.eForcedVentilation,			ePriority := E_BA_Priority.eCritical);
PlantCtrl.AddOperationMode(nOpMode := E_BA_AC_OpMod02.eCentralSwitchOff,			ePriority := E_BA_Priority.eCritical);
PlantCtrl.AddOperationMode(nOpMode := E_BA_AC_OpMod02.eSmokeExtractionProgramm,		ePriority := E_BA_Priority.eLifeSafety);
PlantCtrl.AddOperationMode(nOpMode := E_BA_AC_OpMod02.eSmokeExtractionSupplyAir,	ePriority := E_BA_Priority.eLifeSafety);
PlantCtrl.AddOperationMode(nOpMode := E_BA_AC_OpMod02.eSmokeExtractionExhaustAir,	ePriority := E_BA_Priority.eLifeSafety);
PlantCtrl.AddOperationMode(nOpMode := E_BA_AC_OpMod02.eFire,						ePriority := E_BA_Priority.eLifeSafety);

// Add aggregates:
PlantCtrl.AddAggregate(iReference := PreHtr,	bWaitForProcesses := TRUE,	bWaitForEvents := FALSE, tDelayStepDown := T#0S, tDelayStepUp := T#5S);
PlantCtrl.AddAggregate(iReference := OuADmp,	bWaitForProcesses := FALSE, bWaitForEvents := FALSE, tDelayStepDown := T#2S, tDelayStepUp := T#2S);
PlantCtrl.AddAggregate(iReference := ExhADmp,	bWaitForProcesses := FALSE, bWaitForEvents := FALSE, tDelayStepDown := T#2S, tDelayStepUp := T#2S);
PlantCtrl.AddAggregate(iReference := SuAFan,	bWaitForProcesses := FALSE, bWaitForEvents := FALSE, tDelayStepDown := T#2S, tDelayStepUp := T#2S);
PlantCtrl.AddAggregate(iReference := ExtAFan,	bWaitForProcesses := FALSE, bWaitForEvents := FALSE, tDelayStepDown := T#2S, tDelayStepUp := T#2S);
PlantCtrl.AddAggregate(iReference := Erc,		bWaitForProcesses := FALSE, bWaitForEvents := FALSE, tDelayStepDown := T#0S, tDelayStepUp := T#0S);
PlantCtrl.AddAggregate(iReference := Col,		bWaitForProcesses := FALSE, bWaitForEvents := FALSE, tDelayStepDown := T#0S, tDelayStepUp := T#0S);
PlantCtrl.AddAggregate(iReference := TCasCtrl,	bWaitForProcesses := FALSE, bWaitForEvents := FALSE, tDelayStepDown := T#0S, tDelayStepUp := T#0S);

// Apply aggregate operation modes dependant on corresponding plant operation modes:
// [Controlling aggregates]
// release pre-heater depending on plant operation mode 
PlantCtrl.AssignAggregate1x(nPltOpMode := E_BA_AC_OpMod02.eOff,							iAgg1Ref := PreHtr, nAgg1OpMode := TO_UDINT(FALSE));
PlantCtrl.AssignAggregate1x(nPltOpMode := E_BA_AC_OpMod02.eStep1,						iAgg1Ref := PreHtr, nAgg1OpMode := TO_UDINT(TRUE));
PlantCtrl.AssignAggregate1x(nPltOpMode := E_BA_AC_OpMod02.eStep2,						iAgg1Ref := PreHtr, nAgg1OpMode := TO_UDINT(TRUE));
PlantCtrl.AssignAggregate1x(nPltOpMode := E_BA_AC_OpMod02.eStep3,						iAgg1Ref := PreHtr, nAgg1OpMode := TO_UDINT(TRUE));
PlantCtrl.AssignAggregate1x(nPltOpMode := E_BA_AC_OpMod02.eNightCooling,				iAgg1Ref := PreHtr, nAgg1OpMode := TO_UDINT(FALSE));
PlantCtrl.AssignAggregate1x(nPltOpMode := E_BA_AC_OpMod02.eCoolDownProtection,			iAgg1Ref := PreHtr, nAgg1OpMode := TO_UDINT(TRUE));
PlantCtrl.AssignAggregate1x(nPltOpMode := E_BA_AC_OpMod02.eOverHeatingProtection,		iAgg1Ref := PreHtr, nAgg1OpMode := TO_UDINT(FALSE));
PlantCtrl.AssignAggregate1x(nPltOpMode := E_BA_AC_OpMod02.eFrost,						iAgg1Ref := PreHtr, nAgg1OpMode := TO_UDINT(TRUE));
PlantCtrl.AssignAggregate1x(nPltOpMode := E_BA_AC_OpMod02.eEmergency,					iAgg1Ref := PreHtr, nAgg1OpMode := TO_UDINT(FALSE));
PlantCtrl.AssignAggregate1x(nPltOpMode := E_BA_AC_OpMod02.eAlarm,						iAgg1Ref := PreHtr, nAgg1OpMode := TO_UDINT(FALSE));
PlantCtrl.AssignAggregate1x(nPltOpMode := E_BA_AC_OpMod02.eForcedVentilation,			iAgg1Ref := PreHtr, nAgg1OpMode := TO_UDINT(TRUE));
PlantCtrl.AssignAggregate1x(nPltOpMode := E_BA_AC_OpMod02.eCentralSwitchOff,			iAgg1Ref := PreHtr, nAgg1OpMode := TO_UDINT(FALSE));
PlantCtrl.AssignAggregate1x(nPltOpMode := E_BA_AC_OpMod02.eSmokeExtractionProgramm,		iAgg1Ref := PreHtr, nAgg1OpMode := TO_UDINT(TRUE));
PlantCtrl.AssignAggregate1x(nPltOpMode := E_BA_AC_OpMod02.eSmokeExtractionSupplyAir,	iAgg1Ref := PreHtr, nAgg1OpMode := TO_UDINT(TRUE));
PlantCtrl.AssignAggregate1x(nPltOpMode := E_BA_AC_OpMod02.eSmokeExtractionExhaustAir,	iAgg1Ref := PreHtr, nAgg1OpMode := TO_UDINT(FALSE));
PlantCtrl.AssignAggregate1x(nPltOpMode := E_BA_AC_OpMod02.eFire,						iAgg1Ref := PreHtr, nAgg1OpMode := TO_UDINT(FALSE));

// Apply aggregate operation modes dependant on corresponding plant operation modes:
// [Controlling aggregates]
// release ERC depending on plant operation mode 
PlantCtrl.AssignAggregate1x(E_BA_AC_OpMod02.eOff,							iAgg1Ref := Erc, nAgg1OpMode := TO_UDINT(FALSE));
PlantCtrl.AssignAggregate1x(E_BA_AC_OpMod02.eStep1,							iAgg1Ref := Erc, nAgg1OpMode := TO_UDINT(TRUE));
PlantCtrl.AssignAggregate1x(E_BA_AC_OpMod02.eStep2,							iAgg1Ref := Erc, nAgg1OpMode := TO_UDINT(TRUE));
PlantCtrl.AssignAggregate1x(E_BA_AC_OpMod02.eStep3,							iAgg1Ref := Erc, nAgg1OpMode := TO_UDINT(TRUE));
PlantCtrl.AssignAggregate1x(E_BA_AC_OpMod02.eNightCooling,					iAgg1Ref := Erc, nAgg1OpMode := TO_UDINT(FALSE));
PlantCtrl.AssignAggregate1x(E_BA_AC_OpMod02.eCoolDownProtection,			iAgg1Ref := Erc, nAgg1OpMode := TO_UDINT(TRUE));
PlantCtrl.AssignAggregate1x(E_BA_AC_OpMod02.eOverHeatingProtection,			iAgg1Ref := Erc, nAgg1OpMode := TO_UDINT(TRUE));
PlantCtrl.AssignAggregate1x(E_BA_AC_OpMod02.eFrost,							iAgg1Ref := Erc, nAgg1OpMode := TO_UDINT(TRUE));
PlantCtrl.AssignAggregate1x(E_BA_AC_OpMod02.eEmergency,						iAgg1Ref := Erc, nAgg1OpMode := TO_UDINT(FALSE));
PlantCtrl.AssignAggregate1x(E_BA_AC_OpMod02.eAlarm,							iAgg1Ref := Erc, nAgg1OpMode := TO_UDINT(FALSE));
PlantCtrl.AssignAggregate1x(E_BA_AC_OpMod02.eForcedVentilation,				iAgg1Ref := Erc, nAgg1OpMode := TO_UDINT(TRUE));
PlantCtrl.AssignAggregate1x(E_BA_AC_OpMod02.eCentralSwitchOff,				iAgg1Ref := Erc, nAgg1OpMode := TO_UDINT(FALSE));
PlantCtrl.AssignAggregate1x(E_BA_AC_OpMod02.eSmokeExtractionProgramm,		iAgg1Ref := Erc, nAgg1OpMode := TO_UDINT(TRUE));
PlantCtrl.AssignAggregate1x(E_BA_AC_OpMod02.eSmokeExtractionSupplyAir,		iAgg1Ref := Erc, nAgg1OpMode := TO_UDINT(TRUE));
PlantCtrl.AssignAggregate1x(E_BA_AC_OpMod02.eSmokeExtractionExhaustAir,		iAgg1Ref := Erc, nAgg1OpMode := TO_UDINT(TRUE));
PlantCtrl.AssignAggregate1x(E_BA_AC_OpMod02.eFire,							iAgg1Ref := Erc, nAgg1OpMode := TO_UDINT(FALSE));

// Apply aggregate operation modes dependant on corresponding plant operation modes:
// [Controlling aggregates]
// release cooler depending on plant operation mode 
PlantCtrl.AssignAggregate1x(E_BA_AC_OpMod02.eOff,							iAgg1Ref := Col, nAgg1OpMode := TO_UDINT(FALSE));
PlantCtrl.AssignAggregate1x(E_BA_AC_OpMod02.eStep1,							iAgg1Ref := Col, nAgg1OpMode := TO_UDINT(TRUE));
PlantCtrl.AssignAggregate1x(E_BA_AC_OpMod02.eStep2,							iAgg1Ref := Col, nAgg1OpMode := TO_UDINT(TRUE));
PlantCtrl.AssignAggregate1x(E_BA_AC_OpMod02.eStep3,							iAgg1Ref := Col, nAgg1OpMode := TO_UDINT(TRUE));
PlantCtrl.AssignAggregate1x(E_BA_AC_OpMod02.eNightCooling,					iAgg1Ref := Col, nAgg1OpMode := TO_UDINT(FALSE));
PlantCtrl.AssignAggregate1x(E_BA_AC_OpMod02.eCoolDownProtection,			iAgg1Ref := Col, nAgg1OpMode := TO_UDINT(FALSE));
PlantCtrl.AssignAggregate1x(E_BA_AC_OpMod02.eOverHeatingProtection,			iAgg1Ref := Col, nAgg1OpMode := TO_UDINT(TRUE));
PlantCtrl.AssignAggregate1x(E_BA_AC_OpMod02.eFrost,							iAgg1Ref := Col, nAgg1OpMode := TO_UDINT(FALSE));
PlantCtrl.AssignAggregate1x(E_BA_AC_OpMod02.eEmergency,						iAgg1Ref := Col, nAgg1OpMode := TO_UDINT(FALSE));
PlantCtrl.AssignAggregate1x(E_BA_AC_OpMod02.eAlarm,							iAgg1Ref := Col, nAgg1OpMode := TO_UDINT(FALSE));
PlantCtrl.AssignAggregate1x(E_BA_AC_OpMod02.eForcedVentilation,				iAgg1Ref := Col, nAgg1OpMode := TO_UDINT(TRUE));
PlantCtrl.AssignAggregate1x(E_BA_AC_OpMod02.eCentralSwitchOff,				iAgg1Ref := Col, nAgg1OpMode := TO_UDINT(FALSE));
PlantCtrl.AssignAggregate1x(E_BA_AC_OpMod02.eSmokeExtractionProgramm,		iAgg1Ref := Col, nAgg1OpMode := TO_UDINT(FALSE));
PlantCtrl.AssignAggregate1x(E_BA_AC_OpMod02.eSmokeExtractionSupplyAir,		iAgg1Ref := Col, nAgg1OpMode := TO_UDINT(FALSE));
PlantCtrl.AssignAggregate1x(E_BA_AC_OpMod02.eSmokeExtractionExhaustAir,		iAgg1Ref := Col, nAgg1OpMode := TO_UDINT(FALSE));
PlantCtrl.AssignAggregate1x(E_BA_AC_OpMod02.eFire,							iAgg1Ref := Col, nAgg1OpMode := TO_UDINT(FALSE));

// Apply aggregate operation modes dependant on corresponding plant operation modes:
// [Controlling aggregates]
// [OuADmp]
PlantCtrl.AssignAggregate1x(E_BA_AC_OpMod02.eOff,							iAgg1Ref := OuADmp, nAgg1OpMode := TO_UDINT(FALSE));
PlantCtrl.AssignAggregate1x(E_BA_AC_OpMod02.eStep1,							iAgg1Ref := OuADmp, nAgg1OpMode := TO_UDINT(TRUE)); 
PlantCtrl.AssignAggregate1x(E_BA_AC_OpMod02.eStep2,							iAgg1Ref := OuADmp, nAgg1OpMode := TO_UDINT(TRUE)); 
PlantCtrl.AssignAggregate1x(E_BA_AC_OpMod02.eStep3,							iAgg1Ref := OuADmp, nAgg1OpMode := TO_UDINT(TRUE)); 
PlantCtrl.AssignAggregate1x(E_BA_AC_OpMod02.eNightCooling,					iAgg1Ref := OuADmp, nAgg1OpMode := TO_UDINT(TRUE)); 
PlantCtrl.AssignAggregate1x(E_BA_AC_OpMod02.eCoolDownProtection,			iAgg1Ref := OuADmp, nAgg1OpMode := TO_UDINT(TRUE)); 
PlantCtrl.AssignAggregate1x(E_BA_AC_OpMod02.eOverHeatingProtection,			iAgg1Ref := OuADmp, nAgg1OpMode := TO_UDINT(TRUE)); 
PlantCtrl.AssignAggregate1x(E_BA_AC_OpMod02.eFrost,							iAgg1Ref := OuADmp, nAgg1OpMode := TO_UDINT(FALSE));
PlantCtrl.AssignAggregate1x(E_BA_AC_OpMod02.eEmergency,						iAgg1Ref := OuADmp, nAgg1OpMode := TO_UDINT(FALSE));
PlantCtrl.AssignAggregate1x(E_BA_AC_OpMod02.eAlarm,							iAgg1Ref := OuADmp, nAgg1OpMode := TO_UDINT(FALSE));
PlantCtrl.AssignAggregate1x(E_BA_AC_OpMod02.eForcedVentilation,				iAgg1Ref := OuADmp, nAgg1OpMode := TO_UDINT(TRUE)); 
PlantCtrl.AssignAggregate1x(E_BA_AC_OpMod02.eCentralSwitchOff,				iAgg1Ref := OuADmp, nAgg1OpMode := TO_UDINT(FALSE));
PlantCtrl.AssignAggregate1x(E_BA_AC_OpMod02.eSmokeExtractionProgramm,		iAgg1Ref := OuADmp, nAgg1OpMode := TO_UDINT(TRUE)); 
PlantCtrl.AssignAggregate1x(E_BA_AC_OpMod02.eSmokeExtractionSupplyAir,		iAgg1Ref := OuADmp, nAgg1OpMode := TO_UDINT(TRUE));
PlantCtrl.AssignAggregate1x(E_BA_AC_OpMod02.eSmokeExtractionExhaustAir,		iAgg1Ref := OuADmp, nAgg1OpMode := TO_UDINT(FALSE)); 
PlantCtrl.AssignAggregate1x(E_BA_AC_OpMod02.eFire,							iAgg1Ref := OuADmp, nAgg1OpMode := TO_UDINT(FALSE));

// Apply aggregate operation modes dependant on corresponding plant operation modes:
// [Controlling aggregates]
// [SuAFan]
PlantCtrl.AssignAggregate1x(E_BA_AC_OpMod02.eOff,							iAgg1Ref := SuAFan, nAgg1OpMode := E_BA_3Step.eOff);
PlantCtrl.AssignAggregate1x(E_BA_AC_OpMod02.eStep1,							iAgg1Ref := SuAFan, nAgg1OpMode := E_BA_3Step.eStep1); 
PlantCtrl.AssignAggregate1x(E_BA_AC_OpMod02.eStep2,							iAgg1Ref := SuAFan, nAgg1OpMode := E_BA_3Step.eStep2); 
PlantCtrl.AssignAggregate1x(E_BA_AC_OpMod02.eStep3,							iAgg1Ref := SuAFan, nAgg1OpMode := E_BA_3Step.eStep3); 
PlantCtrl.AssignAggregate1x(E_BA_AC_OpMod02.eNightCooling,					iAgg1Ref := SuAFan, nAgg1OpMode := E_BA_MdltCmd.eOn); 
PlantCtrl.AssignAggregate1x(E_BA_AC_OpMod02.eCoolDownProtection,			iAgg1Ref := SuAFan, nAgg1OpMode := E_BA_MdltCmd.eOn); 
PlantCtrl.AssignAggregate1x(E_BA_AC_OpMod02.eOverHeatingProtection,			iAgg1Ref := SuAFan, nAgg1OpMode := E_BA_MdltCmd.eOn); 
PlantCtrl.AssignAggregate1x(E_BA_AC_OpMod02.eFrost,							iAgg1Ref := SuAFan, nAgg1OpMode := E_BA_MdltCmd.eOff);
PlantCtrl.AssignAggregate1x(E_BA_AC_OpMod02.eEmergency,						iAgg1Ref := SuAFan, nAgg1OpMode := E_BA_MdltCmd.eOff);
PlantCtrl.AssignAggregate1x(E_BA_AC_OpMod02.eAlarm,							iAgg1Ref := SuAFan, nAgg1OpMode := E_BA_MdltCmd.eOff);
PlantCtrl.AssignAggregate1x(E_BA_AC_OpMod02.eForcedVentilation,				iAgg1Ref := SuAFan, nAgg1OpMode := E_BA_MdltCmd.eOn); 
PlantCtrl.AssignAggregate1x(E_BA_AC_OpMod02.eCentralSwitchOff,				iAgg1Ref := SuAFan, nAgg1OpMode := E_BA_MdltCmd.eOff);
PlantCtrl.AssignAggregate1x(E_BA_AC_OpMod02.eSmokeExtractionProgramm,		iAgg1Ref := SuAFan, nAgg1OpMode := E_BA_MdltCmd.eOn); 
PlantCtrl.AssignAggregate1x(E_BA_AC_OpMod02.eSmokeExtractionSupplyAir,		iAgg1Ref := SuAFan, nAgg1OpMode := E_BA_MdltCmd.eOn);
PlantCtrl.AssignAggregate1x(E_BA_AC_OpMod02.eSmokeExtractionExhaustAir,		iAgg1Ref := SuAFan, nAgg1OpMode := E_BA_MdltCmd.eOff); 
PlantCtrl.AssignAggregate1x(E_BA_AC_OpMod02.eFire,							iAgg1Ref := SuAFan, nAgg1OpMode := E_BA_MdltCmd.eOff);

// Apply aggregate operation modes dependant on corresponding plant operation modes:
// [Controlling aggregates]
// [ExhADmp]
PlantCtrl.AssignAggregate1x(E_BA_AC_OpMod02.eOff,							iAgg1Ref := ExhADmp, nAgg1OpMode := TO_UDINT(FALSE));
PlantCtrl.AssignAggregate1x(E_BA_AC_OpMod02.eStep1,							iAgg1Ref := ExhADmp, nAgg1OpMode := TO_UDINT(TRUE)); 
PlantCtrl.AssignAggregate1x(E_BA_AC_OpMod02.eStep2,							iAgg1Ref := ExhADmp, nAgg1OpMode := TO_UDINT(TRUE)); 
PlantCtrl.AssignAggregate1x(E_BA_AC_OpMod02.eStep3,							iAgg1Ref := ExhADmp, nAgg1OpMode := TO_UDINT(TRUE)); 
PlantCtrl.AssignAggregate1x(E_BA_AC_OpMod02.eNightCooling,					iAgg1Ref := ExhADmp, nAgg1OpMode := TO_UDINT(TRUE)); 
PlantCtrl.AssignAggregate1x(E_BA_AC_OpMod02.eCoolDownProtection,			iAgg1Ref := ExhADmp, nAgg1OpMode := TO_UDINT(TRUE)); 
PlantCtrl.AssignAggregate1x(E_BA_AC_OpMod02.eOverHeatingProtection,			iAgg1Ref := ExhADmp, nAgg1OpMode := TO_UDINT(TRUE)); 
PlantCtrl.AssignAggregate1x(E_BA_AC_OpMod02.eFrost,							iAgg1Ref := ExhADmp, nAgg1OpMode := TO_UDINT(FALSE));
PlantCtrl.AssignAggregate1x(E_BA_AC_OpMod02.eEmergency,						iAgg1Ref := ExhADmp, nAgg1OpMode := TO_UDINT(FALSE));
PlantCtrl.AssignAggregate1x(E_BA_AC_OpMod02.eAlarm,							iAgg1Ref := ExhADmp, nAgg1OpMode := TO_UDINT(FALSE));
PlantCtrl.AssignAggregate1x(E_BA_AC_OpMod02.eForcedVentilation,				iAgg1Ref := ExhADmp, nAgg1OpMode := TO_UDINT(TRUE)); 
PlantCtrl.AssignAggregate1x(E_BA_AC_OpMod02.eCentralSwitchOff,				iAgg1Ref := ExhADmp, nAgg1OpMode := TO_UDINT(FALSE));
PlantCtrl.AssignAggregate1x(E_BA_AC_OpMod02.eSmokeExtractionProgramm,		iAgg1Ref := ExhADmp, nAgg1OpMode := TO_UDINT(TRUE)); 
PlantCtrl.AssignAggregate1x(E_BA_AC_OpMod02.eSmokeExtractionSupplyAir,		iAgg1Ref := ExhADmp, nAgg1OpMode := TO_UDINT(FALSE));
PlantCtrl.AssignAggregate1x(E_BA_AC_OpMod02.eSmokeExtractionExhaustAir,		iAgg1Ref := ExhADmp, nAgg1OpMode := TO_UDINT(TRUE)); 
PlantCtrl.AssignAggregate1x(E_BA_AC_OpMod02.eFire,							iAgg1Ref := ExhADmp, nAgg1OpMode := TO_UDINT(FALSE));

// Apply aggregate operation modes dependant on corresponding plant operation modes:
// [Controlling aggregates]
// [ExtAFan]
PlantCtrl.AssignAggregate1x(E_BA_AC_OpMod02.eOff,							iAgg1Ref := ExtAFan, nAgg1OpMode := E_BA_3Step.eOff);
PlantCtrl.AssignAggregate1x(E_BA_AC_OpMod02.eStep1,							iAgg1Ref := ExtAFan, nAgg1OpMode := E_BA_3Step.eStep1); 
PlantCtrl.AssignAggregate1x(E_BA_AC_OpMod02.eStep2,							iAgg1Ref := ExtAFan, nAgg1OpMode := E_BA_3Step.eStep2); 
PlantCtrl.AssignAggregate1x(E_BA_AC_OpMod02.eStep3,							iAgg1Ref := ExtAFan, nAgg1OpMode := E_BA_3Step.eStep3); 
PlantCtrl.AssignAggregate1x(E_BA_AC_OpMod02.eNightCooling,					iAgg1Ref := ExtAFan, nAgg1OpMode := E_BA_MdltCmd.eOn); 
PlantCtrl.AssignAggregate1x(E_BA_AC_OpMod02.eCoolDownProtection,			iAgg1Ref := ExtAFan, nAgg1OpMode := E_BA_MdltCmd.eOn); 
PlantCtrl.AssignAggregate1x(E_BA_AC_OpMod02.eOverHeatingProtection,			iAgg1Ref := ExtAFan, nAgg1OpMode := E_BA_MdltCmd.eOn); 
PlantCtrl.AssignAggregate1x(E_BA_AC_OpMod02.eFrost,							iAgg1Ref := ExtAFan, nAgg1OpMode := E_BA_MdltCmd.eOff);
PlantCtrl.AssignAggregate1x(E_BA_AC_OpMod02.eEmergency,						iAgg1Ref := ExtAFan, nAgg1OpMode := E_BA_MdltCmd.eOff);
PlantCtrl.AssignAggregate1x(E_BA_AC_OpMod02.eAlarm,							iAgg1Ref := ExtAFan, nAgg1OpMode := E_BA_MdltCmd.eOff);
PlantCtrl.AssignAggregate1x(E_BA_AC_OpMod02.eForcedVentilation,				iAgg1Ref := ExtAFan, nAgg1OpMode := E_BA_MdltCmd.eOn); 
PlantCtrl.AssignAggregate1x(E_BA_AC_OpMod02.eCentralSwitchOff,				iAgg1Ref := ExtAFan, nAgg1OpMode := E_BA_MdltCmd.eOff);
PlantCtrl.AssignAggregate1x(E_BA_AC_OpMod02.eSmokeExtractionProgramm,		iAgg1Ref := ExtAFan, nAgg1OpMode := E_BA_MdltCmd.eOn); 
PlantCtrl.AssignAggregate1x(E_BA_AC_OpMod02.eSmokeExtractionSupplyAir,		iAgg1Ref := ExtAFan, nAgg1OpMode := E_BA_MdltCmd.eOff);
PlantCtrl.AssignAggregate1x(E_BA_AC_OpMod02.eSmokeExtractionExhaustAir,		iAgg1Ref := ExtAFan, nAgg1OpMode := E_BA_MdltCmd.eOn); 
PlantCtrl.AssignAggregate1x(E_BA_AC_OpMod02.eFire,							iAgg1Ref := ExtAFan, nAgg1OpMode := E_BA_MdltCmd.eOff);

// Apply aggregate operation modes dependant on corresponding plant operation modes:
// [Controlling aggregates]
// [TCasCtrl]
PlantCtrl.AssignAggregate1x(E_BA_AC_OpMod02.eOff,							TCasCtrl, E_BA_MdltCmd.eOff);
PlantCtrl.AssignAggregate1x(E_BA_AC_OpMod02.eStep1,							TCasCtrl, E_BA_MdltCmd.eOn);
PlantCtrl.AssignAggregate1x(E_BA_AC_OpMod02.eStep2,							TCasCtrl, E_BA_MdltCmd.eOn);
PlantCtrl.AssignAggregate1x(E_BA_AC_OpMod02.eStep3,							TCasCtrl, E_BA_MdltCmd.eOn);
PlantCtrl.AssignAggregate1x(E_BA_AC_OpMod02.eNightCooling,					TCasCtrl, E_BA_MdltCmd.eOff);
PlantCtrl.AssignAggregate1x(E_BA_AC_OpMod02.eCoolDownProtection,			TCasCtrl, E_BA_MdltCmd.eMax);
PlantCtrl.AssignAggregate1x(E_BA_AC_OpMod02.eOverHeatingProtection,			TCasCtrl, E_BA_MdltCmd.eMin);
PlantCtrl.AssignAggregate1x(E_BA_AC_OpMod02.eFrost,							TCasCtrl, E_BA_MdltCmd.eOff);
PlantCtrl.AssignAggregate1x(E_BA_AC_OpMod02.eEmergency,						TCasCtrl, E_BA_MdltCmd.eOff);
PlantCtrl.AssignAggregate1x(E_BA_AC_OpMod02.eAlarm,							TCasCtrl, E_BA_MdltCmd.eOff);
PlantCtrl.AssignAggregate1x(E_BA_AC_OpMod02.eForcedVentilation,				TCasCtrl, E_BA_MdltCmd.eOff);
PlantCtrl.AssignAggregate1x(E_BA_AC_OpMod02.eCentralSwitchOff,				TCasCtrl, E_BA_MdltCmd.eMin);
PlantCtrl.AssignAggregate1x(E_BA_AC_OpMod02.eSmokeExtractionProgramm,		TCasCtrl, E_BA_MdltCmd.eMin);
PlantCtrl.AssignAggregate1x(E_BA_AC_OpMod02.eSmokeExtractionSupplyAir,		TCasCtrl, E_BA_MdltCmd.eOff);
PlantCtrl.AssignAggregate1x(E_BA_AC_OpMod02.eSmokeExtractionExhaustAir,		TCasCtrl, E_BA_MdltCmd.eOff);
PlantCtrl.AssignAggregate1x(E_BA_AC_OpMod02.eFire,							TCasCtrl, E_BA_MdltCmd.eOff);
END_METHOD

METHOD PROTECTED OnInitReferences : BOOL
OnInitReferences := SUPER^.OnInitReferences();

PlantCtrl.Clear();

Init_OffOn();

(*
{error 'Please choose the plants operation mode.'}
// 1) Uncomment one of the following initialization methods to choose operation mode
// 2) Remove the error pragma above

// Init_OffOn();
// Init_OffStep1to3();
*)
END_METHOD

END_FUNCTION_BLOCK

(* stored: Version 1.1.0.1, ProductVersion 3.1.4024.6
   POU FB_BA_AHU_1St_PrHtr_ErcPl_Col: Id {4cfc2b21-c0eb-49a4-9a0d-d04cf2ba3efa}, SpecialFunc None
   Folder Events: Id {b3e2d26a-9ced-4f43-9e36-ff470337d645}
   Folder Initialization: Id {a172b826-54c6-42f9-b2aa-ced024f6e23f}
   Method FB_init: Id {117b0697-8883-45fa-9f9c-d79a25fd0d56}
   Method Init_OffOn: Id {da1fac7c-7cd4-47be-b06a-9e5fccfa1a9c}
   Method Init_OffStep1to3: Id {c132295c-2d43-4156-bdc0-77b502a496b2}
   Method OnInitReferences: Id {52b35c70-60de-402c-890c-9f5353de1d47} *)
